FUNCTION_BLOCK conveyorMotor IMPLEMENTS Imotor
VAR_INPUT
END_VAR
VAR_OUTPUT
END_VAR
VAR
	bStartMotor : BOOL := FALSE;
	bStopMotor : BOOL := TRUE;
	bPauseMotor : BOOL := FALSE;
	eStates : eMotorStates := eMotorStates.firstrun;
	isMotorRunning : BOOL :=  FALSE;
	isError : BOOL := FALSE;
END_VAR

CASE eStates OF
	eMotorStates.firstrun :
		IF bStartMotor THEN
			eStates := eMotorStates.starting;
		END_IF
	eMotorStates.starting:
		IF NOT bStopMotor THEN
			run();
			eStates := eMotorStates.running;
			isMotorRunning := TRUE;
		END_IF
	eMotorStates.running:
		IF bStopMotor THEN
			stop();
			isMotorRunning := FALSE;	
			eStates := eMotorStates.stopped;
		END_IF
		IF bPauseMotor THEN
			eStates := eMotorStates.pause;
		END_IF
	eMotorStates.stopped:
		IF bStartMotor AND NOT bStopMotor THEN
			eStates := eMotorStates.running;
		END_IF
	eMotorStates.pause:
		MpauseMotor();
		eStates := eMotorStates.paused;
	eMotorStates.paused:
		IF bStartMotor AND NOT bStopMotor THEN
			eStates := eMotorStates.running;
		END_IF
		IF  bStopMotor THEN
			eStates := eMotorStates.stopping;
		END_IF
END_CASE


PROPERTY error : BOOL
GET
VAR
	bError : BOOL;
END_VAR
error := isError;
END_GET
SET
isError := error;
END_SET
END_PROPERTY

METHOD MpauseMotor : BOOL
VAR_INPUT
END_VAR
END_METHOD

METHOD run : BOOL
VAR
	bRunMotor: BOOL;
END_VAR
bRunMotor := TRUE;
END_METHOD


PROPERTY running : BOOL
GET
running := isMotorRunning;
END_GET
SET
VAR
	bSimRun : BOOL := False;
END_VAR
isMotorRunning := running;
END_SET
END_PROPERTY

METHOD status : BOOL
VAR
	fbAlarm	: Tc3_EventLogger.FB_TcAlarm;
	bRaiseAlarm	: BOOL;
	bClearAlarm	: BOOL;
	bConfirmAlarm	: BOOL;
	fbSourceInfo	: Tc3_EventLogger.FB_TcSourceInfo;
END_VAR
bRaiseAlarm := TRUE;
END_METHOD

METHOD stop : BOOL
VAR
	bStopM : BOOL;
END_VAR
bStopM := TRUE;
END_METHOD

END_FUNCTION_BLOCK

(* stored: Version 1.1.0.1, ProductVersion 3.1.4024.12
   POU conveyorMotor: Id {921ba089-8039-4ce0-bc80-c9e7a1b5860e}, SpecialFunc None
   Property error: Id {efb640a5-e410-4653-b55f-d74c91aea802}
   Get Get: Id {d1906029-831f-4979-b1b9-2f57c10aea24}
   Set Set: Id {63ce1efd-1b68-4c90-b17a-50f50b2435e5}
   Method MpauseMotor: Id {1d2c00e0-cf18-4bc9-a33b-a67066c79e72}
   Method run: Id {8b17afdc-ad0f-4a5a-808b-4d4e3db20b53}
   Property running: Id {7bbaea36-2752-4125-9591-ec8d8ed77f24}
   Get Get: Id {63f7e8ce-2270-4570-a58a-d3dd0e655874}
   Set Set: Id {d289d6aa-5919-4702-89ec-f8c66608b96e}
   Method status: Id {62b3d55e-d329-4e80-9fff-95eab784407d}
   Method stop: Id {812382a9-ef82-4a69-985d-831d64299f4b} *)
